FUNCTION_BLOCK FB_ProductDataA EXTENDS FB_XP_ProductData IMPLEMENTS I_ProductDataA
VAR
	{attribute 'hide'}	
	stData 	: ST_ProductDataA;
END_VAR

(* It is not necessary to edit anything in this FB. All changes must be made in the "ST_ProductData" structure.
The reason why this FB is not in the CHALET library is that the structure "ST_ProductData" that it contains should be variable.*)

{attribute 'monitoring':='call'}
PROPERTY Data : REFERENCE TO ST_ProductDataA
GET
Data REF= stData;
END_GET
END_PROPERTY

END_FUNCTION_BLOCK

(* stored: Version 1.1.0.1, ProductVersion 3.1.4024.12
   POU FB_ProductDataA: Id {60709667-429a-40f1-9752-df19484c3ac5}, SpecialFunc None
   Property Data: Id {b6e3ed4a-f410-4d25-9730-b9dfa58db76a}
   Get Get: Id {c4675546-e9e3-453c-94ed-8c600b4e1f21} *)
